FUNCTION_BLOCK FB_MoveAbsoluteNC_TestDouble IMPLEMENTS I_MoveABsolute
VAR
    bError : BOOL;
    nErrorID : UDINT := 22000;
END_VAR

PROPERTY Aborted : BOOL
GET
END_GET
END_PROPERTY

PROPERTY Active : BOOL
GET
END_GET
END_PROPERTY

PROPERTY Busy : BOOL
GET
END_GET
END_PROPERTY

PROPERTY CommandMoveAbsolute : BOOL
SET
END_SET
END_PROPERTY

PROPERTY Done : BOOL
GET
END_GET
END_PROPERTY

PROPERTY Error : BOOL
GET
Error := bError;
END_GET
SET
bError := Error;
END_SET
END_PROPERTY

PROPERTY ErrorID : UDINT
GET
ErrorId := nErrorID;
END_GET
SET
nErrorId := ErrorID;
END_SET
END_PROPERTY

PROPERTY Message : T_MAXSTRING
GET
END_GET
END_PROPERTY

METHOD MoveAbsolute
VAR_INPUT
    Position	: LREAL;
    Velocity	: LREAL;
    Acceleration	: LREAL := 0;
    Deceleration	: LREAL := 0;
    Jerk	: LREAL := 0;
    BufferMode	: MC_BufferMode := MC_BufferMode.MC_Aborting;
END_VAR
END_METHOD

{warning 'Add method implementation '}
METHOD MoveAbsoluteDone
END_METHOD

END_FUNCTION_BLOCK

(* stored: Version 1.1.0.1
   POU FB_MoveAbsoluteNC_TestDouble: Id {ee594e6f-53e4-4528-9152-6d9202e100ed}, SpecialFunc None
   Property Aborted: Id {c35c0582-1d5a-4b6e-9c78-63e285fc8bf8}
   Get Get: Id {e123dc24-4ad5-43ff-964d-f052d34939ad}
   Property Active: Id {194dfdf5-ee61-4acf-826d-8d994288cd8c}
   Get Get: Id {edfff653-2b5a-4eae-b74e-ac521933dc03}
   Property Busy: Id {b479a98e-9958-4694-a59a-b0001dec10dd}
   Get Get: Id {3234e5bc-f257-4a74-b140-8484f2499c29}
   Property CommandMoveAbsolute: Id {17406061-5f30-4bfd-8e6d-0a7558c9130d}
   Set Set: Id {8c429de4-e13e-4293-b63d-f8c92c85473d}
   Property Done: Id {d1627f6e-8ac6-41de-9dea-207b8b3ef33f}
   Get Get: Id {7c1f7e30-aa2b-4bbe-9c26-6f1331a8d975}
   Property Error: Id {b643a6d9-c516-44a5-83c7-7a2f58775932}
   Get Get: Id {1ec7862e-a071-43ba-b23f-37b138e357f3}
   Set Set: Id {f687d019-9b82-4ea6-9ead-802882ba9ab0}
   Property ErrorID: Id {1be29702-3d83-4195-abd7-5a87448adc67}
   Get Get: Id {9219ea96-0f16-43ea-9f73-4285d67ee42b}
   Set Set: Id {78a85d56-8cb9-4590-a253-6c09bdfe6d50}
   Property Message: Id {79798b2e-2f42-416d-ac4d-ec72836a1486}
   Get Get: Id {a4461c41-fc0a-49a3-ba5b-0e3e21ad9720}
   Method MoveAbsolute: Id {0f994395-0d64-41f3-8782-3a9802c1d575}
   Method MoveAbsoluteDone: Id {8f9988b0-62d9-4af8-b704-85a4b2006930} *)
